TYPE TYP_HW_L4000_OPC_JOB_CHANGE_OUT :
STRUCT
	Execute AT %Q* : BOOL;
	Filename AT %Q* : STRING;
END_STRUCT
END_TYPE

(* stored: Version 1.1.0.1, ProductVersion 3.1.4024.12
   DUT TYP_HW_L4000_OPC_JOB_CHANGE_OUT: Id {6e818309-2c26-4be6-810f-0ac46f0479a5} *)
